// TwinCAT 3 PLC project Factoryio
// ProgramVersion: 3.1.4026.19
// libraries:
//   Tc2_ModbusSrv, * (Beckhoff Automation GmbH)
//   Tc2_Standard, * (Beckhoff Automation GmbH)
//   Tc2_System, * (Beckhoff Automation GmbH)
// project tree:
//   DUTs/ModbusMap/ ST_ModbusMapCoils.TcDUT (not stored), ST_ModbusMapHoldingRegs.TcDUT (not stored), ST_ModbusMapInputRegs.TcDUT (not stored), ST_ModbusMapInputs.TcDUT
//   DUTs/ ST_FactoryInputs.TcDUT, ST_FactoryOutputs.TcDUT
//   / PlcTask.TcTTO
//   POUs/ FactoryioConnector.TcPOU
// real-time tasks:
//   TASK PlcTaskFactoryioConnector: cycle T#5ms, priority 20, ADS port 350
//   TASK PlcTaskSortieranlage: cycle T#10ms, priority 21, ADS port 351
// variable links:
//   (this object) <-> Sortieranlage/Sortieranlage Instance
//     PlcTask Inputs/FactoryioConnector.stOutputs/bAlarmSiren <-> PlcTask Outputs/GVL_Factory.bAlarmSiren
//     PlcTask Inputs/FactoryioConnector.stOutputs/bBtnResetLight <-> PlcTask Outputs/GVL_Factory.bBtnResetLight
//     PlcTask Inputs/FactoryioConnector.stOutputs/bBtnStartLight <-> PlcTask Outputs/GVL_Factory.bBtnStartLight
//     PlcTask Inputs/FactoryioConnector.stOutputs/bBtnStopLight <-> PlcTask Outputs/GVL_Factory.bBtnStopLight
//     PlcTask Inputs/FactoryioConnector.stOutputs/bConveyorFeed <-> PlcTask Outputs/GVL_Factory.bConveyorFeed
//     PlcTask Inputs/FactoryioConnector.stOutputs/bConveyorForward <-> PlcTask Outputs/GVL_Factory.bConveyorForward
//     PlcTask Inputs/FactoryioConnector.stOutputs/bConveyorLeft <-> PlcTask Outputs/GVL_Factory.bConveyorLeft
//     PlcTask Inputs/FactoryioConnector.stOutputs/bConveyorRight <-> PlcTask Outputs/GVL_Factory.bConveyorRight
//     PlcTask Inputs/FactoryioConnector.stOutputs/bConveyorScale <-> PlcTask Outputs/GVL_Factory.bConveyorScale
//     PlcTask Inputs/FactoryioConnector.stOutputs/bEmitter <-> PlcTask Outputs/GVL_Factory.bEmitter
//     PlcTask Inputs/FactoryioConnector.stOutputs/bSorterLeft <-> PlcTask Outputs/GVL_Factory.bSorterLeft
//     PlcTask Inputs/FactoryioConnector.stOutputs/bSorterRaise <-> PlcTask Outputs/GVL_Factory.bSorterRaise
//     PlcTask Inputs/FactoryioConnector.stOutputs/bSorterRight <-> PlcTask Outputs/GVL_Factory.bSorterRight
//     PlcTask Inputs/FactoryioConnector.stOutputs/bStackLightGreen <-> PlcTask Outputs/GVL_Factory.bStackLightGreen
//     PlcTask Inputs/FactoryioConnector.stOutputs/bStackLightRed <-> PlcTask Outputs/GVL_Factory.bStackLightRed
//     PlcTask Inputs/FactoryioConnector.stOutputs/bStackLightYellow <-> PlcTask Outputs/GVL_Factory.bStackLightYellow
//     PlcTask Inputs/FactoryioConnector.stOutputs/nDispCountForward <-> PlcTask Outputs/GVL_Factory.nDispCountForward
//     PlcTask Inputs/FactoryioConnector.stOutputs/nDispCountLeft <-> PlcTask Outputs/GVL_Factory.nDispCountLeft
//     PlcTask Inputs/FactoryioConnector.stOutputs/nDispCountRight <-> PlcTask Outputs/GVL_Factory.nDispCountRight
//     PlcTask Inputs/FactoryioConnector.stOutputs/nDispWeight <-> PlcTask Outputs/GVL_Factory.nDispWeight
//     PlcTask Inputs/FactoryioConnector.stOutputs/nFactoryCameraPosition <-> PlcTask Outputs/GVL_Factory.nFactoryCameraPosition
//     PlcTask Outputs/FactoryioConnector.stInputs/bBtnReset <-> PlcTask Inputs/GVL_Factory.bBtnReset
//     PlcTask Outputs/FactoryioConnector.stInputs/bBtnStart <-> PlcTask Inputs/GVL_Factory.bBtnStart
//     PlcTask Outputs/FactoryioConnector.stInputs/bBtnStopNC <-> PlcTask Inputs/GVL_Factory.bBtnStopNC
//     PlcTask Outputs/FactoryioConnector.stInputs/bFactoryPaused <-> PlcTask Inputs/GVL_Factory.bFactoryPaused
//     PlcTask Outputs/FactoryioConnector.stInputs/bFactoryReset <-> PlcTask Inputs/GVL_Factory.bFactoryReset
//     PlcTask Outputs/FactoryioConnector.stInputs/bFactoryRunning <-> PlcTask Inputs/GVL_Factory.bFactoryRunning
//     PlcTask Outputs/FactoryioConnector.stInputs/bLbConveyorForwardEntry <-> PlcTask Inputs/GVL_Factory.bLbConveyorForwardEntry
//     PlcTask Outputs/FactoryioConnector.stInputs/bLbConveyorForwardExit <-> PlcTask Inputs/GVL_Factory.bLbConveyorForwardExit
//     PlcTask Outputs/FactoryioConnector.stInputs/bLbConveyorLeftEntry <-> PlcTask Inputs/GVL_Factory.bLbConveyorLeftEntry
//     PlcTask Outputs/FactoryioConnector.stInputs/bLbConveyorLeftExit <-> PlcTask Inputs/GVL_Factory.bLbConveyorLeftExit
//     PlcTask Outputs/FactoryioConnector.stInputs/bLbConveyorRightEntry <-> PlcTask Inputs/GVL_Factory.bLbConveyorRightEntry
//     PlcTask Outputs/FactoryioConnector.stInputs/bLbConveyorRightExit <-> PlcTask Inputs/GVL_Factory.bLbConveyorRightExit
//     PlcTask Outputs/FactoryioConnector.stInputs/bLbScale <-> PlcTask Inputs/GVL_Factory.bLbScale
//     PlcTask Outputs/FactoryioConnector.stInputs/bLbScaleEntry <-> PlcTask Inputs/GVL_Factory.bLbScaleEntry
//     PlcTask Outputs/FactoryioConnector.stInputs/bLbScaleExit <-> PlcTask Inputs/GVL_Factory.bLbScaleExit
//     PlcTask Outputs/FactoryioConnector.stInputs/bSwAuto <-> PlcTask Inputs/GVL_Factory.bSwAuto
//     PlcTask Outputs/FactoryioConnector.stInputs/bSwConveyorFeedOn <-> PlcTask Inputs/GVL_Factory.bSwConveyorFeedOn
//     PlcTask Outputs/FactoryioConnector.stInputs/bSwConveyorForwardOn <-> PlcTask Inputs/GVL_Factory.bSwConveyorForwardOn
//     PlcTask Outputs/FactoryioConnector.stInputs/bSwConveyorLeftOn <-> PlcTask Inputs/GVL_Factory.bSwConveyorLeftOn
//     PlcTask Outputs/FactoryioConnector.stInputs/bSwConveyorRightOn <-> PlcTask Inputs/GVL_Factory.bSwConveyorRightOn
//     PlcTask Outputs/FactoryioConnector.stInputs/bSwConveyorScaleOn <-> PlcTask Inputs/GVL_Factory.bSwConveyorScaleOn
//     PlcTask Outputs/FactoryioConnector.stInputs/bSwEmergStopNC <-> PlcTask Inputs/GVL_Factory.bSwEmergStopNC
//     PlcTask Outputs/FactoryioConnector.stInputs/bSwManual <-> PlcTask Inputs/GVL_Factory.bSwManual
//     PlcTask Outputs/FactoryioConnector.stInputs/fFactoryTimeScale <-> PlcTask Inputs/GVL_Factory.fFactoryTimeScale
//     PlcTask Outputs/FactoryioConnector.stInputs/fScaleWeight <-> PlcTask Inputs/GVL_Factory.fScaleWeight

CONFIGURATION Factoryio
    RESOURCE PLC ON TwinCAT3
        TASK PlcTask(INTERVAL := T#5ms, PRIORITY := 20);
        PROGRAM FactoryioConnector WITH PlcTask : FactoryioConnector;
    END_RESOURCE
END_CONFIGURATION

// ---- DUTs/ModbusMap/ST_ModbusMapInputs.TcDUT
// Factoryio modbus mapping for digital inputs
TYPE ST_ModbusMapInputs:
STRUCT
    // S0 Reset
    bBtnReset: BIT;
    // S1 Start
    bBtnStart: BIT;
    // S2 Stop NC
    bBtnStopNC: BIT;
    // S3 Manual
    bSwManual: BIT;
    // S4 Auto
    bSwAuto: BIT;
    // S5 Emergency stop
    bSwEmergStopNC: BIT;
    // B10 LB: At scale entry
    bLbScaleEntry: BIT;
    // B11 LB: At scale
    bLbScale: BIT;
    // B12 LB: At scale exit
    bLbScaleExit: BIT;
    // B20 LB: At left entry
    bLbConveyorLeftEntry: BIT;
    // B21 LB: At exit left
    bLbConveyorLeftExit: BIT;
    // B30 LB: At forward entry
    bLbConveyorForwardEntry: BIT;
    // B31 LB: At exit front
    bLbConveyorForwardExit: BIT;
    // B40 LB: At right entry
    bLbConveyorRightEntry: BIT;
    // B41 LB: At exit right
    bLbConveyorRightExit: BIT;
    // S100 Band Einlauf ein
    bSwConveyorFeedOn: BIT;
    // S101 Band Auslauf ein
    bSwConveyorForwardOn: BIT;
    // S102 Band Auslauf Links ein
    bSwConveyorLeftOn: BIT;
    // S103 Band Auslauf Rechts ein
    bSwConveyorRightOn: BIT;
    // S104 Band Waage ein
    bSwConveyorScaleOn: BIT;
    // bIn20
    {attribute 'hide'}
    bIn20: BIT;
    // FACTORY I/O (Running)
    bFactoryRunning: BIT;
    // FACTORY I/O (Paused)
    bFactoryPaused: BIT;
    // FACTORY I/O (Reset)
    bFactoryReset: BIT;
END_STRUCT
END_TYPE

// ---- DUTs/ST_FactoryInputs.TcDUT
TYPE ST_FactoryInputs :
STRUCT
    // S0 Reset
    bBtnReset: BIT;
    // S1 Start
    bBtnStart: BIT;
    // S2 Stop NC
    bBtnStopNC: BIT;
    // S3 Manual
    bSwManual: BIT;
    // S4 Auto
    bSwAuto: BIT;
    // S5 Emergency stop
    bSwEmergStopNC: BIT;
    // B10 LB: At scale entry
    bLbScaleEntry: BIT;
    // B11 LB: At scale
    bLbScale: BIT;
    // B12 LB: At scale exit
    bLbScaleExit: BIT;
    // B20 LB: At left entry
    bLbConveyorLeftEntry: BIT;
    // B21 LB: At exit left
    bLbConveyorLeftExit: BIT;
    // B30 LB: At forward entry
    bLbConveyorForwardEntry: BIT;
    // B31 LB: At exit front
    bLbConveyorForwardExit: BIT;
    // B40 LB: At right entry
    bLbConveyorRightEntry: BIT;
    // B41 LB: At exit right
    bLbConveyorRightExit: BIT;
    // S100 Band Einlauf ein
    bSwConveyorFeedOn: BIT;
    // S101 Band Auslauf ein
    bSwConveyorForwardOn: BIT;
    // S102 Band Auslauf Links ein
    bSwConveyorLeftOn: BIT;
    // S103 Band Auslauf Rechts ein
    bSwConveyorRightOn: BIT;
    // S104 Band Waage ein
    bSwConveyorScaleOn: BIT;
    // FACTORY I/O (Running)
    bFactoryRunning: BIT;
    // FACTORY I/O (Paused)
    bFactoryPaused: BIT;
    // FACTORY I/O (Reset)
    bFactoryReset: BIT;
    // Gewicht
    fScaleWeight: REAL;
    // FACTORY I/O (Time Scale)
    fFactoryTimeScale: REAL;
END_STRUCT
END_TYPE

// ---- DUTs/ST_FactoryOutputs.TcDUT
TYPE ST_FactoryOutputs :
STRUCT
    // H0 Reset light
    bBtnResetLight: BIT;
    // H1 Start light
    bBtnStartLight: BIT;
    // H2 Stop light
    bBtnStopLight: BIT;
    // B0 Alarm Siren
    bAlarmSiren: BIT;
    // H20 Signal Light Red
    bStackLightRed: BIT;
    // H21 Signal Light Green
    bStackLightGreen: BIT;
    // H22 Signal Light Yellow
    bStackLightYellow: BIT;
    // M10 Entry conveyor
    bConveyorFeed: BIT;
    // M12 Load scale
    bConveyorScale: BIT;
    // M20 Left conveyor
    bConveyorLeft: BIT;
    // M30 Front conveyor
    bConveyorForward: BIT;
    // M40 Right conveyor
    bConveyorRight: BIT;
    // M50 Send left
    bSorterLeft: BIT;
    // M51 Send forward
    bSorterRaise: BIT;
    // M52 Send right
    bSorterRight: BIT;
    // Emitter
    bEmitter: BIT;
    // Gewicht
    nDispWeight: INT;
    // Left count
    nDispCountLeft: INT;
    // Forward count
    nDispCountForward: INT;
    // Right count
    nDispCountRight: INT;
    // FACTORY I/O (Camera Position)
    nFactoryCameraPosition: INT;
END_STRUCT
END_TYPE

// ---- POUs/FactoryioConnector.TcPOU
PROGRAM FactoryioConnector
VAR
    // IP address of factoryio modbus TCP/IP server
    sFactoryIPAddr: STRING := '127.0.0.1';
    // Port number of factoryio modbus TCP/IP server
    nFactoryTCPPort: UINT := 5502;
    // Modbus slave ID of factoryio modbus TCP/IP server
    nFactoryUnitID: BYTE := 1;
    // Timeout that may not be exceeded by execution of the ADS command
    tConnectionTimeout: TIME := T#2S;

    // Modbus connection to read digital sensors
    fbReadInputs: FB_MBReadInputs;
    // Modbus connection to read analog sensors
    fbReadInputRegs: FB_MBReadInputRegs;
    // Modbus connection to control digital actuators
    fbWriteCoils: FB_MBWriteCoils;
    // Modbus connection to control analog actuators
    fbWriteRegs: FB_MBWriteRegs;

    // Factoryio digital input mapping
    stFactoryioDigitalInputs: ST_ModbusMapInputs;
    // Factoryio analog input mapping
    stFactoryioAnalogInputs: ST_ModbusMapInputRegs;
    // Factoryio digital output mapping
    stFactoryioDigitalOutputs: ST_ModbusMapCoils;
    // Factoryio analog output mapping
    stFactoryioAnalogOutputs: ST_ModbusMapHoldingRegs;

    // Factory Inputs
    stInputs AT %Q*: ST_FactoryInputs;
    // Factory Outputs
    stOutputs AT %I*: ST_FactoryOutputs;
END_VAR

// Read digital sensors
fbReadInputs(
    sIPAddr := sFactoryIPAddr,
    nTCPPort := nFactoryTCPPort,
    nUnitID := nFactoryUnitID,
    nQuantity := 24,
    nMBAddr := 0,
    cbLength := SIZEOF(stFactoryioDigitalInputs),
    pDestAddr := ADR(stFactoryioDigitalInputs),
    tTimeout := tConnectionTimeout
);

IF NOT fbReadInputs.bBusy THEN
    // Assign digital sensors to inputs
    stInputs.bBtnReset := stFactoryioDigitalInputs.bBtnReset;
    stInputs.bBtnStart := stFactoryioDigitalInputs.bBtnStart;
    stInputs.bBtnStopNC := stFactoryioDigitalInputs.bBtnStopNC;
    stInputs.bSwManual := stFactoryioDigitalInputs.bSwManual;
    stInputs.bSwAuto := stFactoryioDigitalInputs.bSwAuto;
    stInputs.bSwEmergStopNC := stFactoryioDigitalInputs.bSwEmergStopNC;
    stInputs.bLbScaleEntry := stFactoryioDigitalInputs.bLbScaleEntry;
    stInputs.bLbScale := stFactoryioDigitalInputs.bLbScale;
    stInputs.bLbScaleExit := stFactoryioDigitalInputs.bLbScaleExit;
    stInputs.bLbConveyorLeftEntry := stFactoryioDigitalInputs.bLbConveyorLeftEntry;
    stInputs.bLbConveyorLeftExit := stFactoryioDigitalInputs.bLbConveyorLeftExit;
    stInputs.bLbConveyorForwardEntry := stFactoryioDigitalInputs.bLbConveyorForwardEntry;
    stInputs.bLbConveyorForwardExit := stFactoryioDigitalInputs.bLbConveyorForwardExit;
    stInputs.bLbConveyorRightEntry := stFactoryioDigitalInputs.bLbConveyorRightEntry;
    stInputs.bLbConveyorRightExit := stFactoryioDigitalInputs.bLbConveyorRightExit;
    stInputs.bSwConveyorFeedOn := stFactoryioDigitalInputs.bSwConveyorFeedOn;
    stInputs.bSwConveyorForwardOn := stFactoryioDigitalInputs.bSwConveyorForwardOn;
    stInputs.bSwConveyorLeftOn := stFactoryioDigitalInputs.bSwConveyorLeftOn;
    stInputs.bSwConveyorRightOn := stFactoryioDigitalInputs.bSwConveyorRightOn;
    stInputs.bSwConveyorScaleOn := stFactoryioDigitalInputs.bSwConveyorScaleOn;
    stInputs.bFactoryRunning := stFactoryioDigitalInputs.bFactoryRunning;
    stInputs.bFactoryPaused := stFactoryioDigitalInputs.bFactoryPaused;
    stInputs.bFactoryReset := stFactoryioDigitalInputs.bFactoryReset;

    // Execute modbus function
    fbReadInputs.bExecute := TRUE;
ELSE
    fbReadInputs.bExecute := FALSE;
END_IF

// Read analog sensors
fbReadInputRegs(
    sIPAddr := sFactoryIPAddr,
    nTCPPort := nFactoryTCPPort,
    nUnitID := nFactoryUnitID,
    nQuantity := 6,
    nMBAddr := 0,
    cbLength := SIZEOF(stFactoryioAnalogInputs),
    pDestAddr := ADR(stFactoryioAnalogInputs),
    tTimeout := tConnectionTimeout
);

IF NOT fbReadInputs.bBusy THEN
    // Assign analog sensors to inputs
    stInputs.fScaleWeight := WORD_TO_REAL(stFactoryioAnalogInputs.fScaleWeight) / 100;
    stInputs.fFactoryTimeScale := WORD_TO_REAL(stFactoryioAnalogInputs.fFactoryTimeScale) / 100;

    // Execute modbus function
    fbReadInputRegs.bExecute := TRUE;
ELSE
    fbReadInputRegs.bExecute := FALSE;
END_IF

// Write digital outputs
fbWriteCoils(
    sIPAddr := sFactoryIPAddr,
    nTCPPort := nFactoryTCPPort,
    nUnitID := nFactoryUnitID,
    nQuantity := 24,
    nMBAddr := 0,
    cbLength := SIZEOF(stFactoryioDigitalOutputs),
    pSrcAddr := ADR(stFactoryioDigitalOutputs),
    tTimeout := tConnectionTimeout
);

IF NOT fbReadInputs.bBusy THEN
    // Assign outputs to digital actuators
    stFactoryioDigitalOutputs.bBtnResetLight := stOutputs.bBtnResetLight;
    stFactoryioDigitalOutputs.bBtnStartLight := stOutputs.bBtnStartLight;
    stFactoryioDigitalOutputs.bBtnStopLight := stOutputs.bBtnStopLight;
    stFactoryioDigitalOutputs.bAlarmSiren := stOutputs.bAlarmSiren;
    stFactoryioDigitalOutputs.bStackLightRed := stOutputs.bStackLightRed;
    stFactoryioDigitalOutputs.bStackLightGreen := stOutputs.bStackLightGreen;
    stFactoryioDigitalOutputs.bStackLightYellow := stOutputs.bStackLightYellow;
    stFactoryioDigitalOutputs.bConveyorFeed := stOutputs.bConveyorFeed;
    stFactoryioDigitalOutputs.bConveyorScale := stOutputs.bConveyorScale;
    stFactoryioDigitalOutputs.bConveyorLeft := stOutputs.bConveyorLeft;
    stFactoryioDigitalOutputs.bConveyorForward := stOutputs.bConveyorForward;
    stFactoryioDigitalOutputs.bConveyorRight := stOutputs.bConveyorRight;
    stFactoryioDigitalOutputs.bSorterLeft := stOutputs.bSorterLeft;
    stFactoryioDigitalOutputs.bSorterRaise := stOutputs.bSorterRaise;
    stFactoryioDigitalOutputs.bSorterRight := stOutputs.bSorterRight;
    stFactoryioDigitalOutputs.bEmitter := stOutputs.bEmitter;

    // Execute modbus function
    fbWriteCoils.bExecute := TRUE;
ELSE
    fbWriteCoils.bExecute := FALSE;
END_IF

// Write analog outputs
fbWriteRegs(
    sIPAddr := sFactoryIPAddr,
    nTCPPort := nFactoryTCPPort,
    nUnitID := nFactoryUnitID,
    nQuantity := 6,
    nMBAddr := 0,
    cbLength := SIZEOF(stFactoryioAnalogOutputs),
    pSrcAddr := ADR(stFactoryioAnalogOutputs),
    tTimeout := tConnectionTimeout
);

IF NOT fbReadInputs.bBusy THEN
    // Assign outputs to analog actuators
    stFactoryioAnalogOutputs.nDispWeight := INT_TO_WORD(stOutputs.nDispWeight);
    stFactoryioAnalogOutputs.nDispCountLeft := INT_TO_WORD(stOutputs.nDispCountLeft);
    stFactoryioAnalogOutputs.nDispCountForward := INT_TO_WORD(stOutputs.nDispCountForward);
    stFactoryioAnalogOutputs.nDispCountRight := INT_TO_WORD(stOutputs.nDispCountRight);
    stFactoryioAnalogOutputs.nFactoryCameraPosition := INT_TO_WORD(stOutputs.nFactoryCameraPosition);

    // Execute modbus function
    fbWriteRegs.bExecute := TRUE;
ELSE
    fbWriteRegs.bExecute := FALSE;
END_IF

END_PROGRAM
